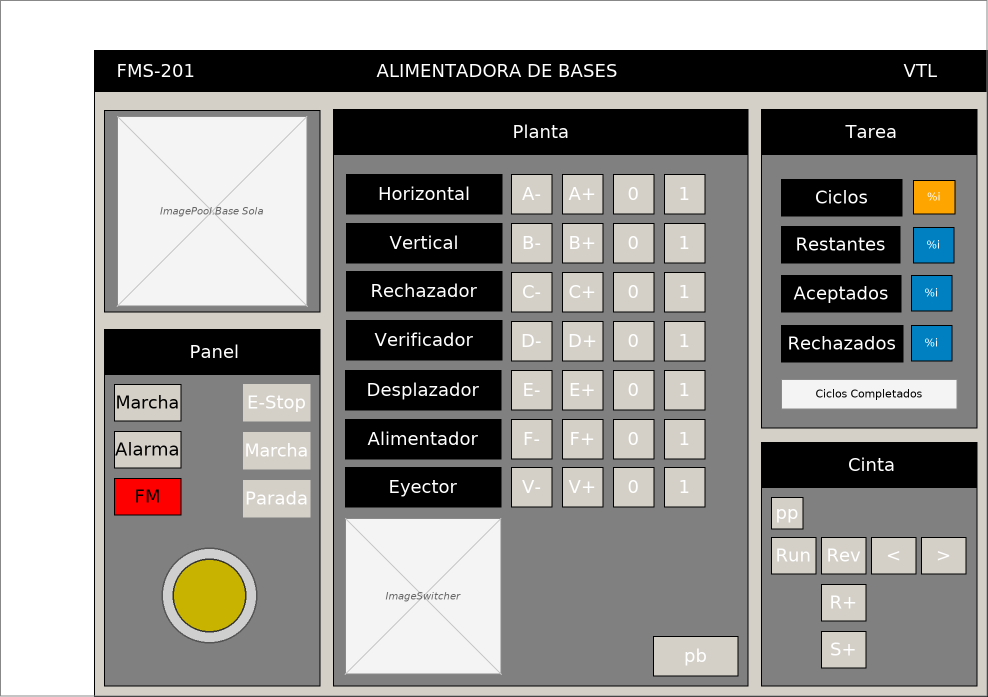
VISUALIZATION Visualization  // 988x697
    Rectangle (94,91 894x606)
    Rectangle (761,154 216x274)
    Rectangle (333,154 415x532)
    Rectangle (333,109 415x45)
    Label (333,111 416x42), "Planta"
    Rectangle (761,109 216x45)
    Label (811,114 121x36), "Tarea"
    Progressbar (781,379 176x30), "Ciclos Completados", variable: MAIN.test_pieza.Aceptados
    RoundedRectangle (346,174 156x40), "Horizontal"
    Textfield (913,180 42x34), "%i", text variable: MAIN.test_pieza.Ciclos
        OnMouseDown: write MAIN.test_pieza.Ciclos via VisuDialogs.Numpad, min 1, max 10
    RoundedRectangle (781,179 121x37), "Ciclos"
    RoundedRectangle (781,226 119x37), "Restantes"
    RoundedRectangle (781,275 120x37), "Aceptados"
    RoundedRectangle (781,325 122x37), "Rechazados"
    Textfield (913,227 41x36), "%i"
    Textfield (911,275 41x36), "%i"
    Textfield (911,325 41x36), "%i"
    RoundedRectangle (562,223 41x40), "B+", colour toggle: MAIN.test_pieza.Descargador_baja
        toggle MAIN.test_pieza.Descargador_baja
    Rectangle (761,487 216x199)
    Rectangle (761,442 216x45)
    Label (811,447 121x36), "Cinta"
    Rectangle (104,110 216x202)
    Rectangle (104,374 216x312)
    Rectangle (104,329 216x45)
    Label (154,334 121x36), "Panel"
    Rectangle (94,50 894x41)
    Label (94,51 893x40), "FMS-201 ALIMENTADORA DE BASES VTL"
    RoundedRectangle (346,223 156x40), "Vertical"
    RoundedRectangle (562,174 41x40), "A+", colour toggle: MAIN.test_pieza.Descargador_adelante
        tap MAIN.test_pieza.Descargador_adelante
    RoundedRectangle (562,272 41x40), "C+", colour toggle: MAIN.test_pieza.Rechazador_adelante
        tap MAIN.test_pieza.Rechazador_adelante
    RoundedRectangle (562,321 41x40), "D+", colour toggle: MAIN.test_pieza.Verificador_baja
        tap MAIN.test_pieza.Verificador_baja
    RoundedRectangle (562,370 41x40), "E+", colour toggle: MAIN.test_pieza.Desplazador_adelante
        tap MAIN.test_pieza.Desplazador_adelante
    RoundedRectangle (562,419 41x40), "F+", colour toggle: MAIN.test_pieza.Alimentador_adelante
        tap MAIN.test_pieza.Alimentador_adelante
        toggle MAIN.test_pieza.Descargador_baja
    RoundedRectangle (562,467 41x40), "V+", colour toggle: MAIN.test_pieza.Eyector_succiona
        toggle MAIN.test_pieza.Eyector_succiona
    RoundedRectangle (346,271 156x40), "Rechazador"
    RoundedRectangle (346,320 156x40), "Verificador"
    RoundedRectangle (345,370 156x40), "Desplazador"
    RoundedRectangle (345,419 156x40), "Alimentador"
    RoundedRectangle (345,467 156x40), "Eyector"
    RoundedRectangle (511,174 41x40), "A-", colour toggle: MAIN.test_pieza.Descargador_atras
        tap MAIN.test_pieza.Descargador_atras
    RoundedRectangle (613,174 41x40), "0", colour toggle: MAIN.test_pieza.Horizontal_descargador_detras
        tap MAIN.test_pieza.Horizontal_descargador_detras
    RoundedRectangle (664,174 41x40), "1", colour toggle: MAIN.test_pieza.Horizontal_descargador_delante
        tap MAIN.test_pieza.Horizontal_descargador_delante
    RoundedRectangle (613,223 41x40), "0", colour toggle: MAIN.test_pieza.Vertical_descargador_arriba
        tap MAIN.test_pieza.Vertical_descargador_arriba
    RoundedRectangle (664,223 41x40), "1", colour toggle: MAIN.test_pieza.Vertical_descargador_abajo
        tap MAIN.test_pieza.Vertical_descargador_abajo
    RoundedRectangle (613,272 41x40), "0"
    RoundedRectangle (613,321 41x40), "0", colour toggle: MAIN.test_pieza.Verificador_arriba
        tap MAIN.test_pieza.Verificador_arriba
    RoundedRectangle (613,370 41x40), "0", colour toggle: MAIN.test_pieza.Desplazador_detras
        tap MAIN.test_pieza.Desplazador_detras
    RoundedRectangle (613,419 41x40), "0", colour toggle: MAIN.test_pieza.Alimentador_detras
        tap MAIN.test_pieza.Alimentador_detras
    RoundedRectangle (613,467 41x40), "0"
    RoundedRectangle (664,272 41x40), "1"
    RoundedRectangle (664,321 41x40), "1", colour toggle: MAIN.test_pieza.Verificador_abajo
        tap MAIN.test_pieza.Verificador_abajo
    RoundedRectangle (664,370 41x40), "1"
    RoundedRectangle (664,419 41x40), "1", colour toggle: MAIN.test_pieza.Alimentador_delante
        tap MAIN.test_pieza.Alimentador_delante
    RoundedRectangle (664,467 41x40), "1", colour toggle: MAIN.test_pieza.Vacio_obtenido_vacuostato_descargador
        tap MAIN.test_pieza.Vacio_obtenido_vacuostato_descargador
    RoundedRectangle (511,223 41x40), "B-"
    RoundedRectangle (511,272 41x40), "C-"
    RoundedRectangle (511,321 41x40), "D-"
    RoundedRectangle (511,370 41x40), "E-"
    RoundedRectangle (511,419 41x40), "F-"
    RoundedRectangle (511,467 41x40), "V-"
    RoundedRectangle (653,636 85x40), "pb", colour toggle: MAIN.test_pieza.Base_en_Alimentador
        tap MAIN.test_pieza.Base_en_Alimentador
    RoundedRectangle (114,478 67x37), "FM", colour toggle: MAIN.test_pieza.Lampara_falta_material
        tap MAIN.test_pieza.Lampara_falta_material
    RoundedRectangle (771,497 32x32), "pp", colour toggle: MAIN.test_pieza.Presencia_pale
        tap MAIN.test_pieza.Presencia_pale
    RoundedRectangle (921,537 45x37), ">", colour toggle: MAIN.test_pieza.Activa_marcha_motor_cinta
        tap MAIN.test_pieza.Activa_marcha_motor_cinta
    RoundedRectangle (871,537 45x37), "<", colour toggle: MAIN.test_pieza.Invierte_marcha_motor_cinta
        toggle MAIN.test_pieza.Invierte_marcha_motor_cinta
    RoundedRectangle (771,537 45x37), "Run", colour toggle: MAIN.test_pieza.Activa_marcha_motor_cinta
    RoundedRectangle (821,537 45x37), "Rev", colour toggle: MAIN.test_pieza.Invierte_marcha_motor_cinta
    RoundedRectangle (821,584 45x37), "R+", colour toggle: MAIN.test_pieza.Retenedor_pale_baja
        tap MAIN.test_pieza.Retenedor_pale_baja
    RoundedRectangle (821,631 45x37), "S+", colour toggle: MAIN.test_pieza.Separador_pale_sube
        tap MAIN.test_pieza.Separador_pale_sube
    RoundedRectangle (243,384 67x37), "E-Stop", colour toggle: MAIN.test_pieza.Pulsador_parada_emergencia
        tap MAIN.test_pieza.Pulsador_parada_emergencia
    RoundedRectangle (243,432 67x37), "Marcha", colour toggle: MAIN.test_pieza.Pulsador_marcha
        tap MAIN.test_pieza.Pulsador_marcha
    RoundedRectangle (243,480 67x37), "Parada", colour toggle: MAIN.test_pieza.Pulsador_parada_NC
        tap MAIN.test_pieza.Pulsador_parada_NC
    RoundedRectangle (114,431 67x37), "Alarma", colour toggle: MAIN.test_pieza.Lampara_alarma
        tap MAIN.test_pieza.Lampara_alarma
    RoundedRectangle (114,384 67x37), "Marcha", colour toggle: MAIN.test_pieza.Lampara_marcha
        tap MAIN.test_pieza.Lampara_marcha
    Image (117,116 190x190), image: ImagePool.Base Sola
    Lamp1 (152,540 115x111), variable: MAIN.test_pieza.Lampara_falta_material, style: Lamp-Lamp1-Yellow
    ImageSwitcher (345,518 156x156), variable: MAIN.test_pieza.pieza_ok, background image: ImagePool.Base OK, image: ImagePool.Base No OK, behaviour: TOGGLE
END_VISUALIZATION

(* stored: Version 1.1.0.1, ProductVersion 3.1.4024.12
   Visu Visualization: Id {fae898df-4a7b-4b14-b77f-db45c2a8e89b} *)
